{attribute 'qualified_only'}
VAR_GLOBAL
	b_recipe_backup	:BOOL;
END_VAR

(* stored: Version 1.1.0.1, ProductVersion 3.1.4024.12
   GVL GVL_Recipe: Id {52970311-9775-474a-a82b-0858d99ac1aa} *)
